// TIA Portal V18 export
FUNCTION_BLOCK "aman_sel_target"   // FB58, FBD
{ S7_Optimized_Access := 'TRUE' }
VERSION : 0.1
// stored: AutoNumber true, IsIECCheckEnabled false, IsRetainMemResEnabled false, MemoryReserve 100, SetENOAutomatically false, UDAEnableTagReadback false
   VAR_INPUT
      allowed : Bool;
      team_unison : Bool;
      team_free : Bool;
      team_override : Bool;
      xbtnAnyMan : Bool;
      xbtnHome : Bool;
      xbtnStepPlus : Bool;
      xbtnStepMinus : Bool;
      execUni : Bool;
      targetUni : Real;
      targetHome : Real;
      targetStep : Real;
      POS : Real;
   END_VAR
   VAR_OUTPUT
      ExecuteSemiAutoManuver : Bool;
      m_auto : Bool;
      m_man : Bool;
      m_override : Bool;
      target : Real;
      execute : Bool;
   END_VAR
   VAR
      auto_allowed : Bool;
      anyBtn : Bool;
      xbtnHome_was : Bool;
      bsuhome { S7_SetPoint := 'True'} : "_ML2_ts_block1_subunit";
      p1Home : Bool;
      q1Home : Bool;
      Q_integer : Int;
      bsu_step_plus { S7_SetPoint := 'True'} : "_ML2_ts_block1_subunit";
      p2StepPlus : Bool;
      q2StepPlus : Bool;
      p3StepMinus : Bool;
      q3StepMinus : Bool;
      bsu_step_minus { S7_SetPoint := 'True'} : "_ML2_ts_block1_subunit";
   END_VAR
   VAR CONSTANT
      Qi0_off : Int := 0;
      Qi1_home : Int := 1;
      Qi2_stepPlus : Int := 2;
      Qi3_stepMinus : Int := 3;
   END_VAR
BEGIN

REGION Network 1
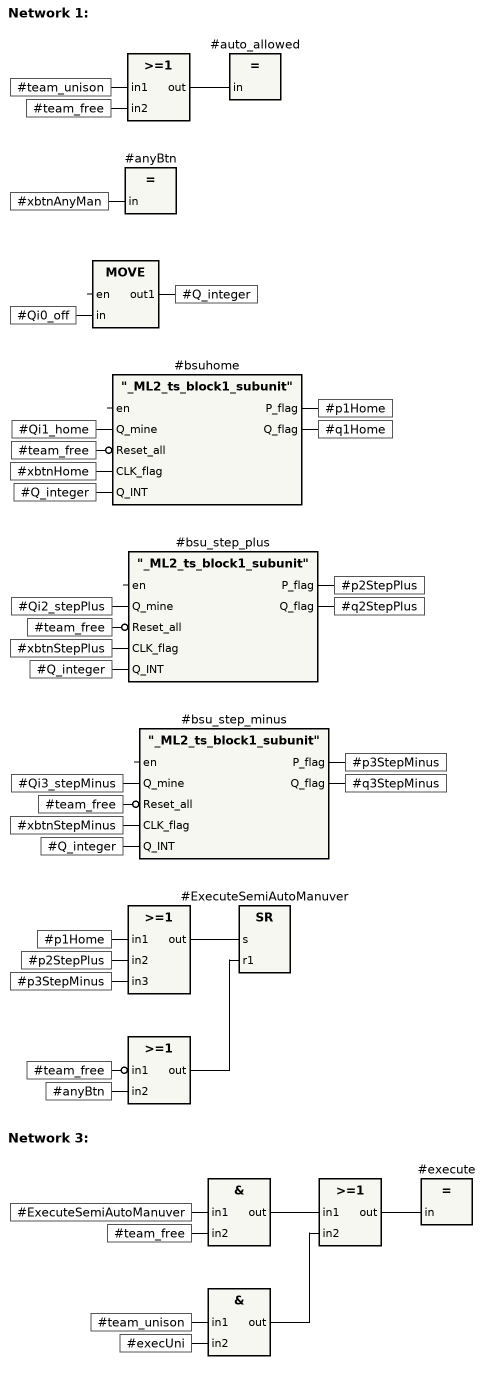
   #auto_allowed := #team_unison OR #team_free;
   #anyBtn := #xbtnAnyMan;
   #Q_integer := #Qi0_off;
   #bsuhome(Q_mine := #Qi1_home,   // "_ML2_ts_block1_subunit"
            Reset_all := NOT #team_free,
            CLK_flag := #xbtnHome,
            Q_INT := #Q_integer,
            P_flag => #p1Home,
            Q_flag => #q1Home);
   #bsu_step_plus(Q_mine := #Qi2_stepPlus,   // "_ML2_ts_block1_subunit"
                  Reset_all := NOT #team_free,
                  CLK_flag := #xbtnStepPlus,
                  Q_INT := #Q_integer,
                  P_flag => #p2StepPlus,
                  Q_flag => #q2StepPlus);
   #bsu_step_minus(Q_mine := #Qi3_stepMinus,   // "_ML2_ts_block1_subunit"
                   Reset_all := NOT #team_free,
                   CLK_flag := #xbtnStepMinus,
                   Q_INT := #Q_integer,
                   P_flag => #p3StepMinus,
                   Q_flag => #q3StepMinus);
   IF #p1Home OR #p2StepPlus OR #p3StepMinus THEN
       #ExecuteSemiAutoManuver := TRUE;   // SR flip-flop
   END_IF;
   IF NOT #team_free OR #anyBtn THEN #ExecuteSemiAutoManuver := FALSE; END_IF;
END_REGION

REGION Network 2 (SCL)
   IF #p1Home THEN
       #target := #targetHome;
   ELSIF #p2StepPlus THEN
       #target := #POS + #targetStep;
   ELSIF #p3StepMinus THEN
       #target := #POS - #targetStep;
   ELSIF #team_unison THEN
       #target := #targetUni;
   END_IF;
   #xbtnHome_was := #xbtnHome;
END_REGION

REGION Network 3
   #execute := (#ExecuteSemiAutoManuver AND #team_free) OR (#team_unison AND #execUni);
END_REGION

REGION Network 4
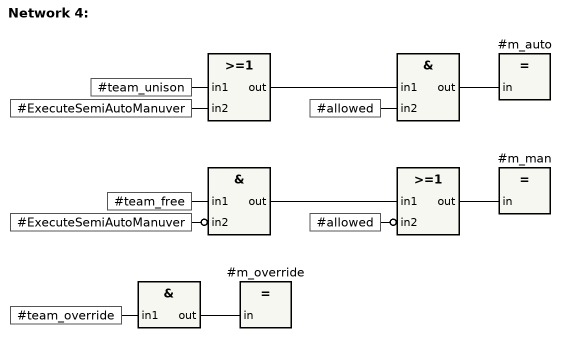
   #m_auto := (#team_unison OR #ExecuteSemiAutoManuver) AND #allowed;
   #m_man := (#team_free AND NOT #ExecuteSemiAutoManuver) OR NOT #allowed;
   #m_override := #team_override;
END_REGION
END_FUNCTION_BLOCK
